{attribute 'qualified_only'}
VAR_GLOBAL
//AH pir data out
	nAH_NeighborRoomsPir_Out		    AT %MB600	: UINT;
	
//AH pir data in
	arrAH_NeighborRoomsPir_In								: ARRAY[1..byNumberOfAH_Neighbors] OF UINT;
	arrAH_NeighborRoomsPir										: ARRAY[1..byNumberOfAH_Neighbors] OF ARRAY[0..15] OF BOOL;
	
//Schneider data out
	nCX8200_State_MB					AT %MB1000		: UINT;
	arrFB_DALIDiagErrorId			(*AT %MW1002*)	: ARRAY[1..SH_Light.DALI_Param.MAX_DALIV2_LINES] OF UDINT;
	arrKL6821InDataStatus				AT %MB1014		: ARRAY[1..SH_Light.DALI_Param.MAX_DALIV2_LINES] OF WORD;
	arrDALILineShrtAddrErr				AT %MB1026		: ARRAY[1..SH_Light.DALI_Param.MAX_DALIV2_LINES] OF UINT;
	EnOceanError						AT %MB1038		: UINT;
	nTotalEnergy10kWh						AT %MB1040		: UINT;
	nMaxControlGearOperatingHours 	    AT %MB1042		: UINT;
	uiPirOffDelayTimeAllRooms_MB   AT %MB1044   : UINT := 30;
END_VAR
VAR_GLOBAL CONSTANT
	byNumberOfAH_Neighbors									: BYTE := 25;
END_VAR

(*
AH2-2 pirsignaler = arrAH_NeighborRoomsPir[1]
	---------- KOPI fra A_AHNeighborRoomsPirOut i AH2-2 ----------
	GVL_AHDataModbus.nAH_NeighborRoomsPir_Out.0		:= P_Gang_2_244A.bPirActive_MB;
	GVL_AHDataModbus.nAH_NeighborRoomsPir_Out.1		:= P_Gang_7_201.bPirActive_MB;
*)

(*
AH4-2 pirsignaler = arrAH_NeighborRoomsPir[2]
	---------- KOPI fra A_AHNeighborRoomsPirOut i AH4-2 ----------
	GVL_AHDataModbus.nAH_NeighborRoomsPir_Out.0		:= P_Gang_3_109.bPirActive_MB;
*)

//3 etage:
(*AH2-3 
GVL_AHDataModbus.nAH_NeighborRoomsPir_Out.0 := P_Gang_2_344.bPirActive_MB;
GVL_AHDataModbus.nAH_NeighborRoomsPir_Out.1 := P_Gang_7_301.bPirActive_MB;
//GVL_AHDataModbus.nAH_NeighborRoomsPir_Out.2 := P_Rum_2_349.bPirActive_MB;
//GVL_AHDataModbus.nAH_NeighborRoomsPir_Out.1 := P_Gang_2_341.bPirActive_MB;*)

(*AH3-3
GVL_AHDataModbus.nAH_NeighborRoomsPir_Out.0 := P_Gang_3_364.bPirActive_MB;
GVL_AHDataModbus.nAH_NeighborRoomsPir_Out.1 := P_Gang_3_309.bPirActive_MB;
GVL_AHDataModbus.nAH_NeighborRoomsPir_Out.2 := P_Gang_2_350.bPirActive_MB;*)

(* stored: Version 1.1.0.1
   GVL GVL_AHDataModbus: Id {f5902466-9696-4cef-8487-6320c343acc6} *)
